TYPE Pixel : UDINT; END_TYPE

(* stored: Version 1.1.0.1, ProductVersion 3.1.4024.15
   DUT Pixel: Id {b4985355-4d8a-457c-8dd2-2e186652966b} *)
